{attribute addProperty BoxType "KL6401-0002"}
{attribute addProperty Id "Channel_1Channel_172861D000"}
{attribute addProperty CRC "1632467114"}
{attribute addProperty SizeInBites "0"}
{attribute addProperty SizeInBytes "0"}
TYPE KL_614D78AA :
STRUCT
	{attribute addProperty Name "Channel_1"}
	Channel_1 : Channel_172861D0;
END_STRUCT
END_TYPE

(* stored: Version 1.2.0.0, ProductVersion 3.1.4024.9
   DUT KL_614D78AA: Id {456483fb-d1b0-4ecb-aa52-46d65543244d} *)
